FUNCTION_BLOCK GreenMasterBaseParameters
VAR_IN_OUT
	GreenMaster: GreenMasterBase;
END_VAR
VAR_INPUT
	System: SystemParametersFB;
	Regulation: RegulationParametersFB;
	Alarm: AlarmParameters;
	IO: IoParametersFB;
END_VAR
VAR_OUTPUT
END_VAR
VAR
END_VAR

System(Parameters := THIS^);
Regulation(Parameters := THIS^);
IO(GreenMaster := GreenMaster, Parameters := THIS^);

END_FUNCTION_BLOCK

(* stored: Version 1.1.0.1, ProductVersion 3.1.4022.18
   POU GreenMasterBaseParameters: Id {4f104a97-9854-4cb1-aeb3-f00bd259eb43}, SpecialFunc None *)
